Fanuc KAREL source: kt00529.KL

PROGRAM KT00529
%STACKSIZE=65535
%PRIORITY=65535
%NOLOCKGROUP
VAR
P1 : XYZWPREXT
P2 : JOINTPOS9
OUT : POSITION
BEGIN
P1.X=1.0
-- UNRESOLVED_PC line 9 opcodes [49 7E 49 7E 60 4A] marker_code=20
END KT00529
